% RSLogix 500 project SENSOR_CALIBRATION.RSS, saved by version 8.30.00.16 %
PROJECT "UNTITLED"    % processor: Bul.1763 MicroLogix 1100 Series B %

PROGRAM FILES
  LAD 2 "MAIN"  5 rungs
  LAD 3 "I/O"  5 rungs
  LAD 4 "CONTROL"  9 rungs
  LAD 5 "COMPUTE"  7 rungs

DATA FILES
  O0 OUTPUT  7 elements
  I1 INPUT  13 elements
  S2 STATUS  66 elements
  B3 BINARY  3 elements
  T4 TIMER  4 elements
  C5 COUNTER  2 elements
  R6 CONTROL  1 elements
  N7 INTEGER  11 elements
  F8 FLOAT  1 elements

LADDER 2 "MAIN"
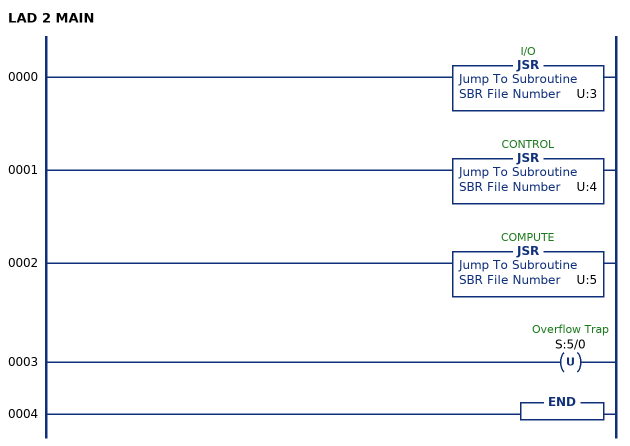
% Rung: 0 %
SOR JSR U:3 EOR
%   U:3  "I/O" %
% Rung: 1 %
SOR JSR U:4 EOR
%   U:4  "CONTROL" %
% Rung: 2 %
SOR JSR U:5 EOR
%   U:5  "COMPUTE" %
% Rung: 3 %
SOR OTU S:5/0 EOR
%   S:5/0  "Overflow Trap" %
% Rung: 4 %
SOR END EOR

LADDER 3 "I/O"
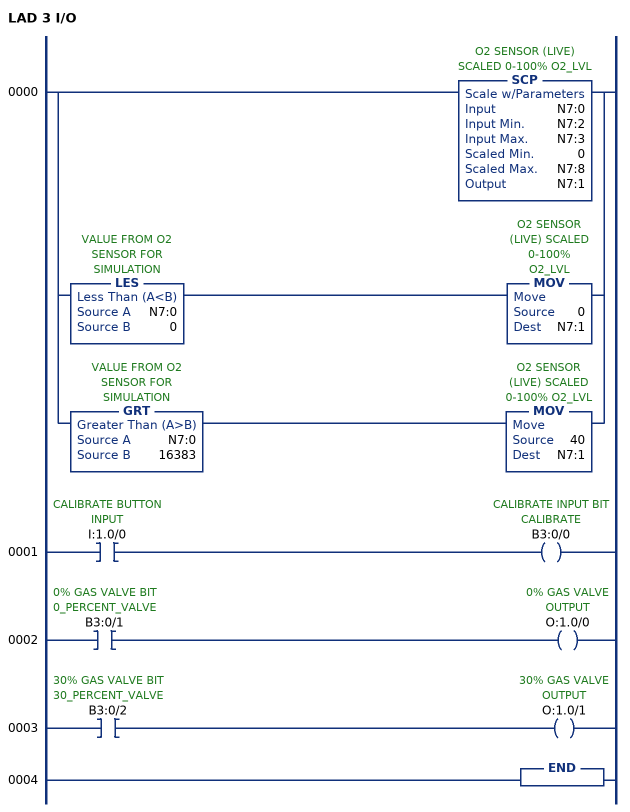
% Rung: 0 %
SOR BST SCP N7:0 N7:2 N7:3 0 N7:8 N7:1 NXB LES N7:0 0 MOV 0 N7:1 NXB GRT N7:0 16383 MOV 40 N7:1 BND EOR
%   N7:0  "VALUE FROM O2 SENSOR FOR SIMULATION" %
%   N7:2  "INPUT MINIMUM CALIBRATED (DEFAULT WAS 0)" %
%   N7:3  "INPUT MAXIMUM CALIBRATED (DEFAULT WAS 16383)" %
%   N7:8  MAX_CONCENTRATION  "MAXIMUM PERMISSIBLE CONCENTRATION" %
%   N7:1  O2_LVL  "O2 SENSOR (LIVE) SCALED 0-100%" %
% Rung: 1 %
SOR XIC I:1.0/0 OTE B3:0/0 EOR
%   I:1.0/0  "CALIBRATE BUTTON INPUT" %
%   B3:0/0  CALIBRATE  "CALIBRATE INPUT BIT" %
% Rung: 2 %
SOR XIC B3:0/1 OTE O:1.0/0 EOR
%   B3:0/1  0_PERCENT_VALVE  "0% GAS VALVE BIT" %
%   O:1.0/0  "0% GAS VALVE OUTPUT" %
% Rung: 3 %
SOR XIC B3:0/2 OTE O:1.0/1 EOR
%   B3:0/2  30_PERCENT_VALVE  "30% GAS VALVE BIT" %
%   O:1.0/1  "30% GAS VALVE OUTPUT" %
% Rung: 4 %
SOR END EOR

LADDER 4 "CONTROL"
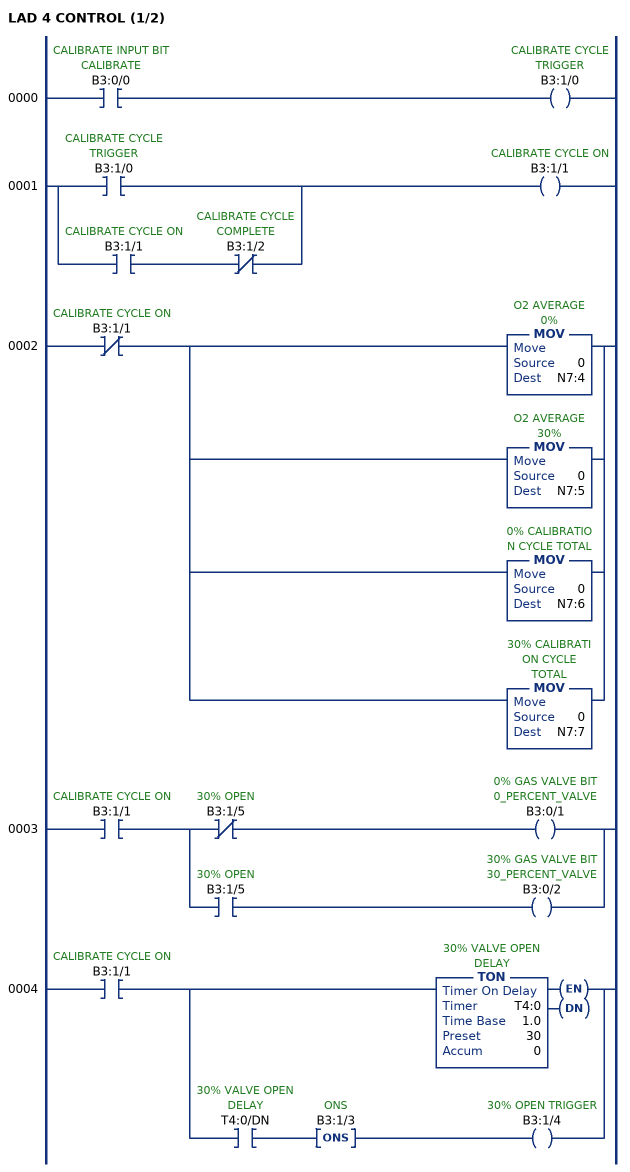
% Rung: 0 %
SOR XIC B3:0/0 OTE B3:1/0 EOR
%   B3:0/0  CALIBRATE  "CALIBRATE INPUT BIT" %
%   B3:1/0  "CALIBRATE CYCLE TRIGGER" %
% Rung: 1 %
SOR BST XIC B3:1/0 NXB XIC B3:1/1 XIO B3:1/2 BND OTE B3:1/1 EOR
%   B3:1/0  "CALIBRATE CYCLE TRIGGER" %
%   B3:1/1  "CALIBRATE CYCLE ON" %
%   B3:1/2  "CALIBRATE CYCLE COMPLETE" %
% Rung: 2 %
SOR XIO B3:1/1 BST MOV 0 N7:4 NXB MOV 0 N7:5 NXB MOV 0 N7:6 NXB MOV 0 N7:7 BND EOR
%   B3:1/1  "CALIBRATE CYCLE ON" %
%   N7:4  "O2 AVERAGE 0%" %
%   N7:5  "O2 AVERAGE 30%" %
%   N7:6  "0% CALIBRATION CYCLE TOTAL" %
%   N7:7  "30% CALIBRATION CYCLE TOTAL" %
% Rung: 3 %
SOR XIC B3:1/1 BST XIO B3:1/5 OTE B3:0/1 NXB XIC B3:1/5 OTE B3:0/2 BND EOR
%   B3:1/1  "CALIBRATE CYCLE ON" %
%   B3:1/5  "30% OPEN" %
%   B3:0/1  0_PERCENT_VALVE  "0% GAS VALVE BIT" %
%   B3:0/2  30_PERCENT_VALVE  "30% GAS VALVE BIT" %
% Rung: 4 %
SOR XIC B3:1/1 BST TON T4:0 1.0 30 0 NXB XIC T4:0/DN ONS B3:1/3 OTE B3:1/4 BND EOR
%   B3:1/1  "CALIBRATE CYCLE ON" %
%   T4:0  "30% VALVE OPEN DELAY" %
%   T4:0/DN  "30% VALVE OPEN DELAY" %
%   B3:1/3  "ONS" %
%   B3:1/4  "30% OPEN TRIGGER" %

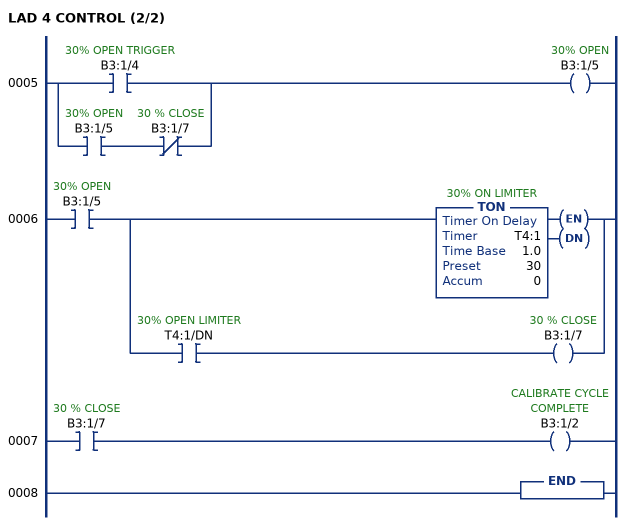
% Rung: 5 %
SOR BST XIC B3:1/4 NXB XIC B3:1/5 XIO B3:1/7 BND OTE B3:1/5 EOR
%   B3:1/4  "30% OPEN TRIGGER" %
%   B3:1/5  "30% OPEN" %
%   B3:1/7  "30 % CLOSE" %
% Rung: 6 %
SOR XIC B3:1/5 BST TON T4:1 1.0 30 0 NXB XIC T4:1/DN OTE B3:1/7 BND EOR
%   B3:1/5  "30% OPEN" %
%   T4:1  "30% ON LIMITER" %
%   T4:1/DN  "30% OPEN LIMITER" %
%   B3:1/7  "30 % CLOSE" %
% Rung: 7 %
SOR XIC B3:1/7 OTE B3:1/2 EOR
%   B3:1/7  "30 % CLOSE" %
%   B3:1/2  "CALIBRATE CYCLE COMPLETE" %
% Rung: 8 %
SOR END EOR

LADDER 5 "COMPUTE"
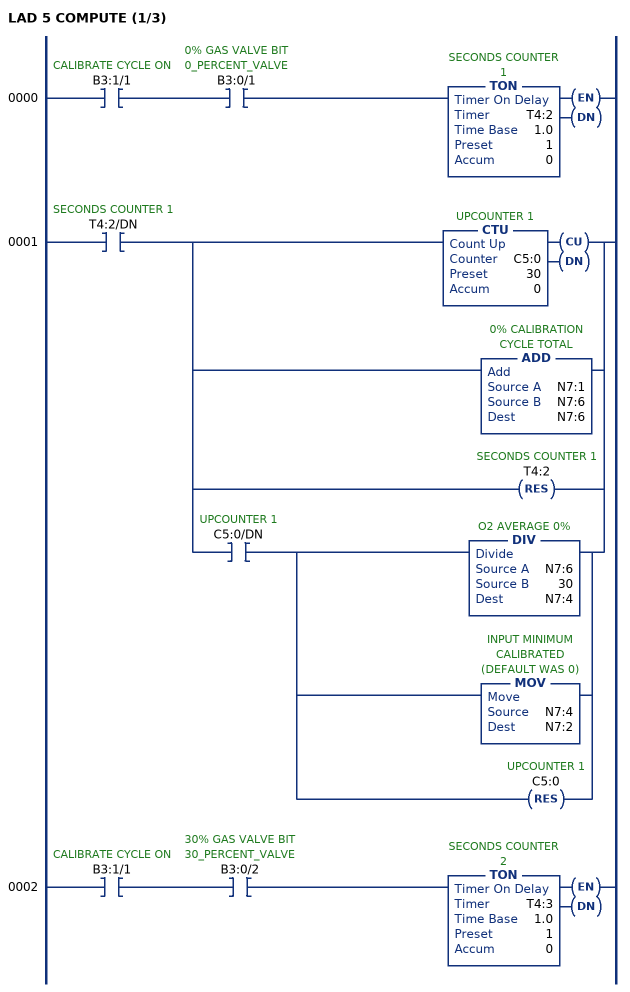
% Rung: 0 %
SOR XIC B3:1/1 XIC B3:0/1 TON T4:2 1.0 1 0 EOR
%   B3:1/1  "CALIBRATE CYCLE ON" %
%   B3:0/1  0_PERCENT_VALVE  "0% GAS VALVE BIT" %
%   T4:2  "SECONDS COUNTER 1" %
% Rung: 1 %
SOR XIC T4:2/DN BST CTU C5:0 30 0 NXB ADD N7:1 N7:6 N7:6 NXB RES T4:2 NXB XIC C5:0/DN BST DIV N7:6 30 N7:4 NXB MOV N7:4 N7:2 NXB RES C5:0 BND BND EOR
%   T4:2/DN  "SECONDS COUNTER 1" %
%   C5:0  "UPCOUNTER 1" %
%   N7:1  O2_LVL  "O2 SENSOR (LIVE) SCALED 0-100%" %
%   N7:6  "0% CALIBRATION CYCLE TOTAL" %
%   T4:2  "SECONDS COUNTER 1" %
%   C5:0/DN  "UPCOUNTER 1" %
%   N7:4  "O2 AVERAGE 0%" %
%   N7:2  "INPUT MINIMUM CALIBRATED (DEFAULT WAS 0)" %
% Rung: 2 %
SOR XIC B3:1/1 XIC B3:0/2 TON T4:3 1.0 1 0 EOR
%   B3:1/1  "CALIBRATE CYCLE ON" %
%   B3:0/2  30_PERCENT_VALVE  "30% GAS VALVE BIT" %
%   T4:3  "SECONDS COUNTER 2" %

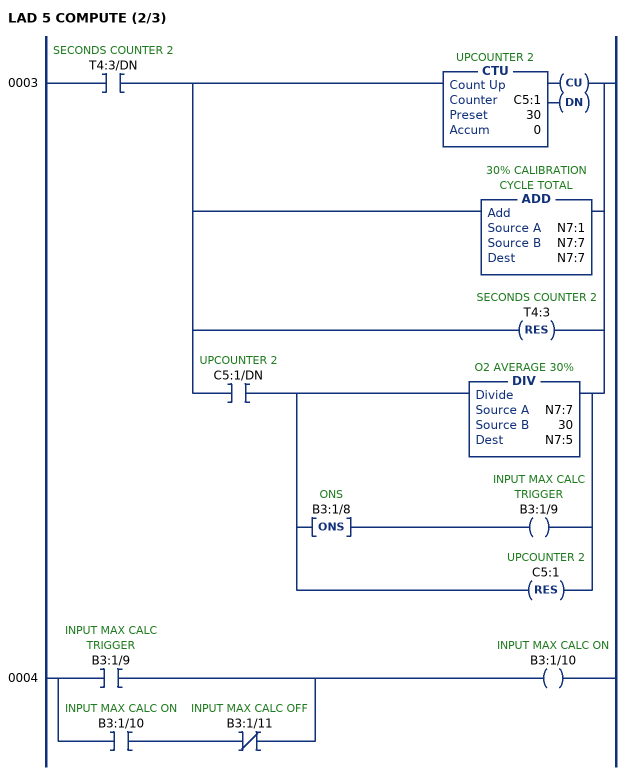
% Rung: 3 %
SOR XIC T4:3/DN BST CTU C5:1 30 0 NXB ADD N7:1 N7:7 N7:7 NXB RES T4:3 NXB XIC C5:1/DN BST DIV N7:7 30 N7:5 NXB ONS B3:1/8 OTE B3:1/9 NXB RES C5:1 BND BND EOR
%   T4:3/DN  "SECONDS COUNTER 2" %
%   C5:1  "UPCOUNTER 2" %
%   N7:1  O2_LVL  "O2 SENSOR (LIVE) SCALED 0-100%" %
%   N7:7  "30% CALIBRATION CYCLE TOTAL" %
%   T4:3  "SECONDS COUNTER 2" %
%   C5:1/DN  "UPCOUNTER 2" %
%   N7:5  "O2 AVERAGE 30%" %
%   B3:1/8  "ONS" %
%   B3:1/9  "INPUT MAX CALC TRIGGER" %
% Rung: 4 %
SOR BST XIC B3:1/9 NXB XIC B3:1/10 XIO B3:1/11 BND OTE B3:1/10 EOR
%   B3:1/9  "INPUT MAX CALC TRIGGER" %
%   B3:1/10  "INPUT MAX CALC ON" %
%   B3:1/11  "INPUT MAX CALC OFF" %

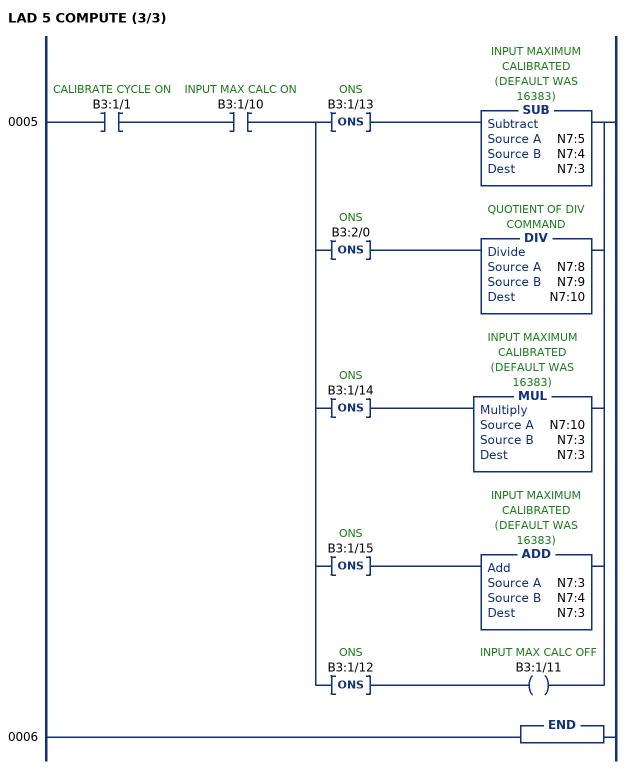
% Rung: 5 %
SOR XIC B3:1/1 XIC B3:1/10 BST ONS B3:1/13 SUB N7:5 N7:4 N7:3 NXB ONS B3:2/0 DIV N7:8 N7:9 N7:10 NXB ONS B3:1/14 MUL N7:10 N7:3 N7:3 NXB ONS B3:1/15 ADD N7:3 N7:4 N7:3 NXB ONS B3:1/12 OTE B3:1/11 BND EOR
%   B3:1/1  "CALIBRATE CYCLE ON" %
%   B3:1/10  "INPUT MAX CALC ON" %
%   B3:1/13  "ONS" %
%   N7:5  "O2 AVERAGE 30%" %
%   N7:4  "O2 AVERAGE 0%" %
%   N7:3  "INPUT MAXIMUM CALIBRATED (DEFAULT WAS 16383)" %
%   B3:2/0  "ONS" %
%   N7:8  MAX_CONCENTRATION  "MAXIMUM PERMISSIBLE CONCENTRATION" %
%   N7:9  CALI_GAS_CONC  "CALIBRATION GAS CONCENTRATION" %
%   N7:10  "QUOTIENT OF DIV COMMAND" %
%   B3:1/14  "ONS" %
%   B3:1/15  "ONS" %
%   B3:1/12  "ONS" %
%   B3:1/11  "INPUT MAX CALC OFF" %
% Rung: 6 %
SOR END EOR

OTHER DOCUMENTED ADDRESSES
  B3:1/6  "ONS"
  I:2.0/0  "O2 SENSOR INPUT"

COMMENTS NOT ATTACHED TO A CURRENT RUNG
  N7:3: CALIBRATION FROMULA:-
    ((O2-MAX CONCENTRATION / O2-CALIBRATION GAS CONCENTRATION) * (O2 TEST GAS AVERAGE - O2 ZERO AVERAGE)) + O2 ZERO AVERAGE

DATA TABLE (non-zero values as saved)
DATA T4
% .PRE .ACC %
% T4:0 % 30 0
% T4:1 % 30 0
% T4:2 % 1 0
% T4:3 % 1 0
DATA C5
% .PRE .ACC %
% C5:0 % 30 0
% C5:1 % 30 0
DATA N7
% N7:0 % 0 0 0 16383 0 0 0 0 40 30
